FUNCTION_BLOCK Print
  (* Version 1.0, 2005-07-05, Goran Cengic, Chalmers *)
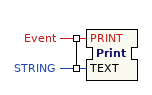
  EVENT_INPUT
    PRINT WITH TEXT;
  END_EVENT
  VAR_INPUT
    TEXT : STRING;
  END_VAR
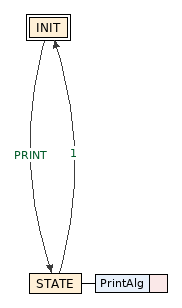
  EC_STATES
    INIT;
    STATE : PrintAlg;
  END_STATES
  EC_TRANSITIONS
    INIT TO STATE := PRINT;
    STATE TO INIT := 1;
  END_TRANSITIONS
  ALGORITHM PrintAlg IN Java:
System.out.println(TEXT);
  END_ALGORITHM
END_FUNCTION_BLOCK
